{attribute 'qualified_only'}
{attribute 'strict'}
TYPE E_WHITESPACE_LOCATION :
(
	Both := 0,
	Start,
	End
);
END_TYPE

(* stored: Version 1.1.0.1, ProductVersion 3.1.4024.4
   EnumerationTextList E_WHITESPACE_LOCATION: Id {9d6f670b-f439-486e-bf56-b056829de42f} *)
